// TIA Portal V16 export
// export: Created 2023-03-29T11:03:38.6328714Z, ExportSetting WithDefaults, DisplayName Totally Integrated Automation Portal, DisplayVersion V16 Update 6, DisplayName TIA Portal Version Control Interface, DisplayVersion V16 Update 2, DisplayName TIA Portal Openness, DisplayVersion V16 Update 6, DisplayName STEP 7 Professional, DisplayVersion V16 Update 6, DisplayName STEP 7 Safety, DisplayVersion V16, DisplayName WinCC Advanced, DisplayVersion V16 Update 6
DATA_BLOCK "operating_mode_select_aut-man_DB"   // DB53
AUTHOR : rtecmer
VERSION : 0.1
// stored: AutoNumber true, DBAccessibleFromOPCUA true, InstanceOfName operating_mode_select_aut-man, InstanceOfType FB
"operating_mode_select_aut-man"
   // VAR
   //    setTrig_Z1 : Bool;
   //    setTrig_Z2 : Bool;
   //    setTrig_Z3 : Bool;
   //    setTrig_Z4 : Bool;
   //    setTrig_Z5 : Bool;
   //    setTrig_Z6 : Bool;
   //    setTrig_Z7 : Bool;
   //    setTrig_Z8 : Bool;
   //    setTrig_Z9 : Bool;
   //    setTrig_Z10 : Bool;
   //    set_aut_man_Z1 : Bool;
   //    set_aut_man_Z2 : Bool;
   //    set_aut_man_Z3 : Bool;
   //    set_aut_man_Z4 : Bool;
   //    set_aut_man_Z5 : Bool;
   //    set_aut_man_Z6 : Bool;
   //    set_aut_man_Z7 : Bool;
   //    set_aut_man_Z8 : Bool;
   //    set_aut_man_Z9 : Bool;
   //    set_aut_man_Z10 : Bool;
   // END_VAR
BEGIN
END_DATA_BLOCK
